PROGRAM P06_LidFeeder
VAR_INPUT
	IbLidFeederDragHomingSensor 			AT %I*  : BOOL;				// Czujnik bazowania
	IbLidFeederDragUpSensor 			 	AT %I*  : BOOL;				// Czujnik
	IbLidFeederDragDownSensor 				AT %I*  : BOOL;				// Czujnik
	IbLidFeederDragLeadBefore1UpSensor 		AT %I*  : BOOL;				// Czujnik
	IbLidFeederUpSensor1 					AT %I*	: BOOL; 								// Czujnik pozycji górnej ssawki podajnika platynek
	IbLidFeederUpSensor2 					AT %I*	: BOOL;
	IbLidFeederDownSensor1 					AT %I*	: BOOL;								
	IbLidFeederDownSensor2 					AT %I*	: BOOL;								
	IbLidFeederLowLevelSensor1  			AT %I* 	: BOOL;	
	IbLidFeederLowLevelSensor2  			AT %I* 	: BOOL;
	IbLidFeederFormPositioning1HideSensor			AT %I*	: BOOL; 
	IbLidFeederFormPositioning2HideSensor			AT %I*	: BOOL;
	IbLidFeederFirstFormSensorBeforeDrag			AT %I*	:BOOL;
	IbLidFeederSuckerSensor 				AT %I*	: BOOL;
	IbLidFeeder2SuckerSensor 				AT %I*	: BOOL;  
	bMovetoEndPositionLidFeeder				:BOOL;	
	QbLidFeederDragActuator                	  		: BOOL;				// Siłownikiem przeciągania (1 faza)					

END_VAR
VAR
	//Podajnik platynek
	fbLidFeeder										: FB_LidFeeder; 						// Blok sterowania podajnikiem platynek
	eLidFeederState									: E_Station; 							// Stan pracy podajnika platynek			
	eLidFeederRunningState							: E_LidFeederState; 					// Stan pracy podajnika platynek
	fbLidFeederState								: FB_State; 

	//Podajnik platynek 2
	fbLidFeeder2									: FB_LidFeeder; 						// Blok sterowania podajnikiem platynek
	eLidFeeder2State								: E_Station; 							// Stan pracy podajnika platynek			
	eLidFeeder2RunningState							: E_LidFeederState; 					// Stan pracy podajnika platynek
	fbLidFeeder2State								: FB_State; 

	QbLidFeederBlockActuator 				AT %Q*	: BOOL;  		// Blokada 
	
	// WEJŚCIA I WYJŚCIA SPRZĘTOWE 1
	QbLidFeeder_FeederActuator1						: BOOL; 				(*Pneu*) 		// Sterowanie zaworem podajnika platynek na wyspie zaworowej
	QbLidFeeder_FeederActuator2						: BOOL; 				(*Pneu*) 		// Sterowanie zaworem podajnika platynek na wyspie zaworowej
	QbLidFeeder_HeaterActuator						: BOOL;  				(*Pneu*) 		// Sterowanie zaworem grzałki platynek na wyspie zaworowej
	QbLidFeeder_SuckerActuator 				AT %Q*	: BOOL; 								// Sterowanie zaworem ssawki platynek na wyspie zaworowej
	QbLidFeederHeaterPWMOut 				AT %Q*	: BOOL; 								// Wyjście sterujące grzałką podajnika platynek
	

	AIbLidFeederHeaterTempCVSensor 			AT %I*	: INT; 									// Wartość aktualnej temperatury grzałki podajnika platynek
	IbLidFeederTempSensorFailure 			AT %I*	: BOOL; 								// Informacja o uszkodzeniu czujnika temperatury grzałki podajnika platynek
	QbLidFeeder_HeightMotorUp 				AT %Q*	: BOOL;									// Sterowanie silnikiem podnosnika stacji w górę 
	QbLidFeeder_HeightMotorDown 			AT %Q*	: BOOL;									//Sterowanie silnikiem podnosnika stacji w dół
	IbLidFeederHeightEncoderPulse  			AT %I* 	: BOOL;									// Wejście impulsów enkodera podnośnika platynek regulacji wysokości 
									// Czujnik niskiego pozimu platynek	
	
	// WEJŚCIA I WYJŚCIA SPRZĘTOWE 2		
	QbLidFeeder2_FeederActuator1					: BOOL; 				(*Pneu*) 		// Sterowanie zaworem podajnika platynek na wyspie zaworowej
	QbLidFeeder2_FeederActuator2					: BOOL; 				(*Pneu*) 		// Sterowanie zaworem podajnika platynek na wyspie zaworowej
	QbLidFeeder2_HeaterActuator						: BOOL;  				(*Pneu*) 		// Sterowanie zaworem grzałki platynek na wyspie zaworowej
	QbLidFeeder2_SuckerActuator 			AT %Q*	: BOOL; 								// Sterowanie zaworem ssawki platynek na wyspie zaworowej
	QbLidFeeder2HeaterPWMOut 				AT %Q*	: BOOL; 								// Wyjście sterujące grzałką podajnika platynek
	IbLidFeeder2UpSensor1 					AT %I*	: BOOL; 								// Czujnik pozycji górnej ssawki podajnika platynek
	IbLidFeeder2DownSensor1 				AT %I*	: BOOL;								
	IbLidFeeder2DownSensor2 				AT %I*	: BOOL;								
									// Czujnik zassania platynki
	AIbLidFeeder2HeaterTempCVSensor 		AT %I*	: INT; 									// Wartość aktualnej temperatury grzałki podajnika platynek
	IbLidFeeder2TempSensorFailure 			AT %I*	: BOOL; 								// Informacja o uszkodzeniu czujnika temperatury grzałki podajnika platynek
										// Czujnik niskiego pozimu platynek
	
	//Vasyl 24.10.25 Aktualizacja enkodera
	IbLidFeederHeightEncoderSetCDone		AT %I*: BOOL;	
	IudiLidFeederHeightEncoderCV         	AT %I*: UDINT; 	
	QbLidFeederHeightEncoderSetC 			AT %Q*: BOOL;		
	QudiLidFeederHeightEncoderSetCV       	AT %Q*: UDINT; 	
	
	tofLidFeederEnable								: TOF;
	tonLidFeederEnable								: TON;
	rtEnable										: R_TRIG;

	tonLidFeederCatchSensorClosed					: TON;
                	
	bTemp											: BOOL;
	bSimulation										: BOOL;
	
	bLidFeederWarning1								: BOOL;
	bLidFeederWarning2								: BOOL;
	
	//PRZECIAGANIE
	eLidFeederDragStation							: E_Station;
	eLidFeederDragRunningStation					: E_DragStationState;
	fbLidFeederDragState							: FB_State;
	fbLidFeederDragStation							: FB_FormsDragStepper;

	tofLidFeederDragStationEnable					: TOF;	
	
	//WEJSCIA I WYJSCIA SPRZETOWE
	QbLidFeederDragLeadBefore1Actuator        		: BOOL;				// Siłownikiem prowadzenia przed 1(1 faza)
	QbLidFeederDragLeadBefore2Actuator        		: BOOL;				// Siłownikiem prowadzenia przed 1(1 faza)
	
	
	IbLidFeederDragLeadBefore2UpSensor 				AT %I*  : BOOL;				// Czujnik
	
	bLidFeederUp									: BOOL;				//Podnoszenie podajników do góry
	
	
	//Chwytak formatek
	fbLidFeederFormPositioning						: FB_Gate;				// Bloczek obsługi bandy
	IbLidFeederFormPositioningUpSensor				AT %I*	: BOOL; 		// 
	QbLidFeederFormPositioningActuator 				: BOOL;  		



	
	bTestManual: BOOL;
END_VAR

//QbLidFeederBlockActuator	:= (GVL.eLidFeederPackageState[1].bFormPresent AND GVL.bFormTransportersDispencerCmdStart) OR 
//							   (GVL.eLidFeederPackageState[2].bFormPresent AND GVL.bFormTransportersDispencerCmdStart);

IF P00_PackML.fbPMLModeManager.eModeStatus = Tc3_PackML.E_PMLUnitMode.ePMLUnitMode_AUTOMATIC AND tofLidFeederEnable.Q THEN
	
	QbLidFeederBlockActuator :=	P00_PackML.fbPMLAuto.ePMLState = Tc3_PackML.E_PMLState.ePMLState_EXECUTE OR 
								P00_PackML.fbPMLAuto.ePMLState = Tc3_PackML.E_PMLState.ePMLState_STOPPING OR 
								P00_PackML.fbPMLAuto.ePMLState = Tc3_PackML.E_PMLState.ePMLState_STARTING;
								
ELSIF P00_PackML.fbPMLModeManager.eModeStatus = Tc3_PackML.E_PMLUnitMode.ePMLUnitMode_MANUAL THEN
	
	QbLidFeederBlockActuator	:= P06_LidSealer.fbLidSealer.bBlockActuator OR P06_LidSealer.fbLidSealer2.bBlockActuator OR VIS.bLidFeeder1ManualHeaterAct OR VIS.bLidFeeder2ManualHeaterAct OR
			VIS.bLidFeeder1Run OR VIS.bLidFeeder2Run OR VIS.bLidFeederEnableShow;
	
END_IF

bLidFeederUp	:= GVL_IO.IbEmergencyStopButton0Pressed OR GVL_IO.IbEmergencyStopButton1Pressed OR GVL_IO.IbEmergencyStopButton2Pressed OR {warning 'PI odkomentować'}
				   GVL_IO.IbEmergencyStopButton3Pressed OR GVL_IO.IbEmergencyStopButton4Pressed OR IbTurnTableEmergencyStopButtonPressed OR (*IbPucksInserterEmergencyStopButton0Pressed OR*) IbPucksInserterEmergencyStopButton1Pressed
				   OR P07_ROPP.IbROPPEmergencyStopButton0Pressed OR P07_ROPP.IbROPPEmergencyStopButton1Pressed 
				AND (QbLidFeeder_HeaterActuator OR QbLidFeeder2_HeaterActuator);
							   
ACT_LidFeeder();
ACT_LidFeeder2();
ACT_LidFeederDragStation();
a_LidFeederFormPositioning();
aLidFeederWarnings();

//GENEROWANIE STANU STACJI DO WIZKI
fbLidFeederState(
	eState 					:= eLidFeederState , 
	bRun 					:= VIS.bLidFeeder1PrepareRun OR VIS.bLidFeeder1Run,	
	eLidFeederRunningState 	:= eLidFeederRunningState , 
	sStateDesc				=> VIS.sLidFeeder1State,
	iState					=> VIS.iLidFeeder1State	);
	
fbLidFeeder2State(
	eState 					:= eLidFeeder2State , 
	bRun 					:= VIS.bLidFeeder2PrepareRun OR VIS.bLidFeeder2Run,	
	eLidFeederRunningState 	:= eLidFeeder2RunningState , 
	sStateDesc				=> VIS.sLidFeeder2State,
	iState					=> VIS.iLidFeeder2State	);
	
(* BAZOWANIE - ZMIAN*)
tonLidFeederEnable(IN := fbLidFeeder.bEnable, PT := T#2S); (*Dodany ton bo Wizka zjebnie wgrywa zmienne, najpierw włacza Enabla a potem dopiero wybiera recepture*)
rtEnable(CLK := tonLidFeederEnable.Q, Q=>);
IF rtEnable.Q AND (P00_PackML.fbPMLAuto.ePMLState = Tc3_PackML.E_PMLState.ePMLState_IDLE OR 
   P00_PackML.fbPMLAuto.ePMLState = Tc3_PackML.E_PMLState.ePMLState_EXECUTE) THEN
    VIS.bLidFeederHeightSet 		:= TRUE;
ELSIF (fbLidFeeder.eState = E_Station.eHomingDone AND fbLidFeeder2.eState = E_Station.eHomingDone)OR VIS.bErrorOccure THEN
    VIS.bLidFeederHeightSet 		:= FALSE;
END_IF
(*KONIEC BAZOWANIE - ZMIANA*)

//PRZEPISYWANIE POMIARÓW
VIS.lrLidFeeder1HeaterTempCV	:= (INT_TO_LREAL(AIbLidFeederHeaterTempCVSensor)/10);
VIS.lrLidFeeder2HeaterTempCV	:= (INT_TO_LREAL(AIbLidFeeder2HeaterTempCVSensor)/10);

//SYMULACJA CZUJNIKÓW IGLIC

//Opoznienie wyłączanie enabla
tofLidFeederEnable(IN:= VIS.bLidFeederEnableShow, PT:=T#2S);

//KASOWANIE ROZKAZÓW CYKLI
IF fbLidFeeder.bCycleDone AND GVL.bManualMode THEN
	VIS.bLidFeeder1PrepareRun 		:= FALSE;
	VIS.bLidFeeder1Run 			:= FALSE;
END_IF
IF fbLidFeeder2.bCycleDone AND GVL.bManualMode THEN
	VIS.bLidFeeder2PrepareRun 		:= FALSE;
	VIS.bLidFeeder2Run 			:= FALSE;
END_IF

IF bSimulation THEN
	IF fbLidFeeder.eState = E_Station.eReady AND fbLidFeeder2.eState = E_Station.eReady THEN
		VIS.bLidFeeder1PrepareRun	:= TRUE;
		VIS.bLidFeeder2PrepareRun	:= TRUE;
	END_IF
	IF fbLidFeeder.eState = E_Station.eRunning AND fbLidFeeder2.eState = E_Station.eRunning THEN
		
		IF (VIS.bLidFeeder1PrepareRun AND NOT VIS.bLidFeeder1Run AND IbLidFeederDownSensor1) AND
		   (VIS.bLidFeeder2PrepareRun AND NOT VIS.bLidFeeder2Run AND IbLidFeeder2DownSensor1) THEN		
			VIS.bLidFeeder1Run 	:= TRUE;
			VIS.bLidFeeder2Run 	:= TRUE;		
	
		END_IF
	END_IF
	
	IF fbLidFeeder.bCycleDone AND fbLidFeeder2.bCycleDone THEN
		
		VIS.bLidFeeder1PrepareRun	:= FALSE;
		VIS.bLidFeeder2PrepareRun	:= FALSE;
		VIS.bLidFeeder1Run 		:= FALSE;
		VIS.bLidFeeder2Run 		:= FALSE;
		
	END_IF
END_IF

(*
{warning: 'Sprawdzic działanie czujnika niskiego poziomu - kiedy stan wysoki'}

//Ostrzeżenia Podajnik 1 
GVL.LidFeederWarning[0].sDescription			:= 'Niski poziom platynek podajnik 1';

IF bLidFeederWarning1 AND NOT GVL.LidFeederWarning[0].bWarning THEN
	
	GVL.LidFeederWarning[0].bWarning			:= TRUE;
	
ELSIF NOT bLidFeederWarning1 AND GVL.LidFeederWarning[0].bAcknowledge THEN
	
	GVL.LidFeederWarning[0].bWarning			:= FALSE;
	GVL.LidFeederWarning[0].bAcknowledge		:= FALSE;
	//GvlVisualization.uliWarningAcknowledge.4 	:= FALSE;
	
ELSIF GVL.LidFeederWarning[0].bAcknowledge THEN
{warning: 'Sprawdzic potwierdzenie warningu tutaj i wewnatrz bloczka gdy zmieni sie stan czujnika '}	
	bLidFeederWarning1							:= FALSE;
	GVL.LidFeederWarning[0].bAcknowledge		:= TRUE;
	
END_IF

//Ostrzeżenia Podajnik 2 
GVL.LidFeederWarning[1].sDescription			:= 'Niski poziom platynek podajnik 2';

IF bLidFeederWarning2 AND NOT GVL.LidFeederWarning[1].bWarning THEN
	
	GVL.LidFeederWarning[1].bWarning			:= TRUE;
	
ELSIF NOT bLidFeederWarning2 AND GVL.LidFeederWarning[1].bAcknowledge THEN
	
	GVL.LidFeederWarning[1].bWarning			:= FALSE;
	GVL.LidFeederWarning[1].bAcknowledge		:= FALSE;
	//GvlVisualization.uliWarningAcknowledge.4 	:= FALSE;
	
ELSIF GVL.LidFeederWarning[1].bAcknowledge THEN
	
	bLidFeederWarning2							:= FALSE;	
	GVL.LidFeederWarning[1].bAcknowledge		:= TRUE;
	
END_IF
*)

//Przeciąganie
tofLidFeederDragStationEnable(IN:= VIS.bLidFeederDragingStationEnableShow, PT:= T#2S);

ACTION a_LidFeederFormPositioning:
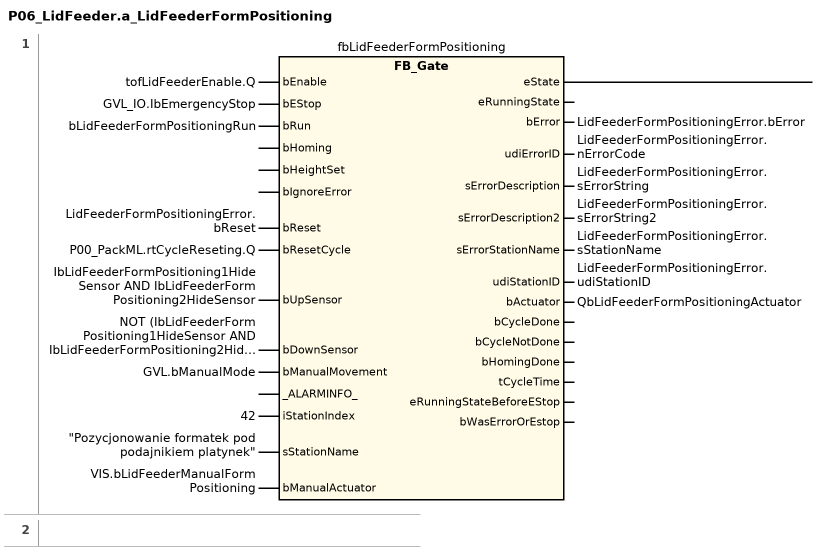
// NETWORK 1
fbLidFeederFormPositioning(
    bEnable := tofLidFeederEnable.Q,
    bEStop := GVL_IO.IbEmergencyStop,
    bRun := bLidFeederFormPositioningRun,
    bReset := LidFeederFormPositioningError.bReset,
    bResetCycle := P00_PackML.rtCycleReseting.Q,
    bUpSensor := IbLidFeederFormPositioning1HideSensor AND IbLidFeederFormPositioning2HideSensor,
    bDownSensor := NOT (IbLidFeederFormPositioning1HideSensor AND IbLidFeederFormPositioning2HideSensor),
    bManualMovement := GVL.bManualMode,
    iStationIndex := 42,
    sStationName := "Pozycjonowanie formatek pod podajnikiem platynek",
    bManualActuator := VIS.bLidFeederManualFormPositioning,
    bError => LidFeederFormPositioningError.bError,
    udiErrorID => LidFeederFormPositioningError.nErrorCode,
    sErrorDescription => LidFeederFormPositioningError.sErrorString,
    sErrorDescription2 => LidFeederFormPositioningError.sErrorString2,
    sErrorStationName => LidFeederFormPositioningError.sStationName,
    udiStationID => LidFeederFormPositioningError.udiStationID,
    bActuator => QbLidFeederFormPositioningActuator); // FB_Gate

// NETWORK 2
END_ACTION

ACTION ACT_LidFeeder:
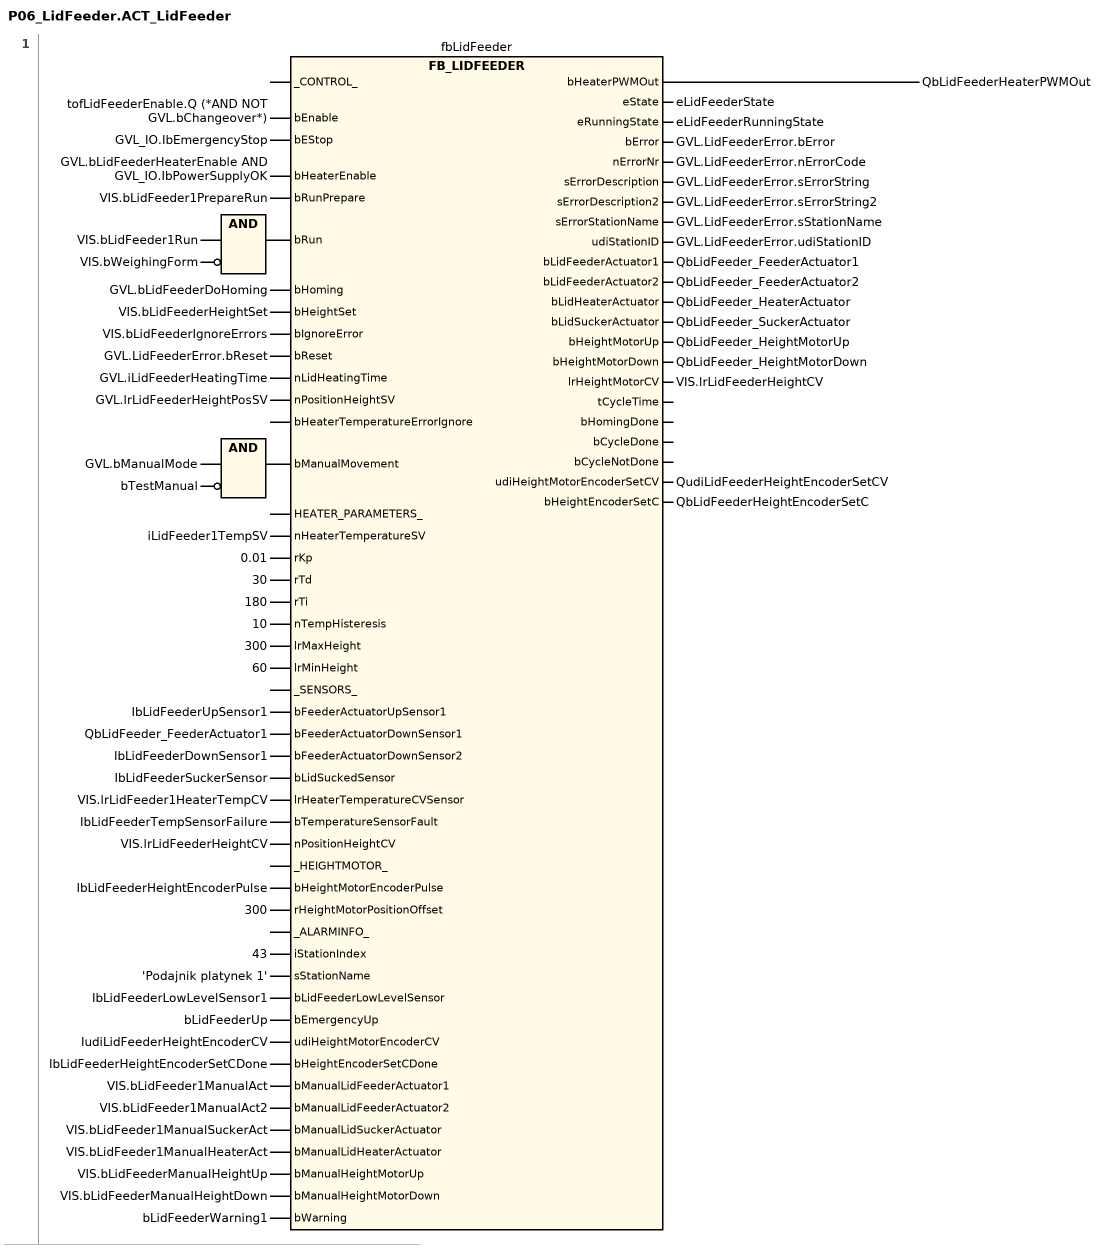
// NETWORK 1
fbLidFeeder(
    bEnable := tofLidFeederEnable.Q (*AND NOT GVL.bChangeover*),
    bEStop := GVL_IO.IbEmergencyStop,
    bHeaterEnable := GVL.bLidFeederHeaterEnable AND GVL_IO.IbPowerSupplyOK,
    bRunPrepare := VIS.bLidFeeder1PrepareRun,
    bRun := VIS.bLidFeeder1Run AND NOT VIS.bWeighingForm,
    bHoming := GVL.bLidFeederDoHoming,
    bHeightSet := VIS.bLidFeederHeightSet,
    bIgnoreError := VIS.bLidFeederIgnoreErrors,
    bReset := GVL.LidFeederError.bReset,
    nLidHeatingTime := GVL.iLidFeederHeatingTime,
    nPositionHeightSV := GVL.lrLidFeederHeightPosSV,
    bManualMovement := GVL.bManualMode AND NOT bTestManual,
    nHeaterTemperatureSV := iLidFeeder1TempSV,
    rKp := 0.01,
    rTd := 30,
    rTi := 180,
    nTempHisteresis := 10,
    lrMaxHeight := 300,
    lrMinHeight := 60,
    bFeederActuatorUpSensor1 := IbLidFeederUpSensor1,
    bFeederActuatorDownSensor1 := QbLidFeeder_FeederActuator1,
    bFeederActuatorDownSensor2 := IbLidFeederDownSensor1,
    bLidSuckedSensor := IbLidFeederSuckerSensor,
    lrHeaterTemperatureCVSensor := VIS.lrLidFeeder1HeaterTempCV,
    bTemperatureSensorFault := IbLidFeederTempSensorFailure,
    nPositionHeightCV := VIS.lrLidFeederHeightCV,
    bHeightMotorEncoderPulse := IbLidFeederHeightEncoderPulse,
    rHeightMotorPositionOffset := 300,
    iStationIndex := 43,
    sStationName := 'Podajnik platynek 1',
    bLidFeederLowLevelSensor := IbLidFeederLowLevelSensor1,
    bEmergencyUp := bLidFeederUp,
    udiHeightMotorEncoderCV := IudiLidFeederHeightEncoderCV,
    bHeightEncoderSetCDone := IbLidFeederHeightEncoderSetCDone,
    bManualLidFeederActuator1 := VIS.bLidFeeder1ManualAct,
    bManualLidFeederActuator2 := VIS.bLidFeeder1ManualAct2,
    bManualLidSuckerActuator := VIS.bLidFeeder1ManualSuckerAct,
    bManualLidHeaterActuator := VIS.bLidFeeder1ManualHeaterAct,
    bManualHeightMotorUp := VIS.bLidFeederManualHeightUp,
    bManualHeightMotorDown := VIS.bLidFeederManualHeightDown,
    bWarning := bLidFeederWarning1,
    eState => eLidFeederState,
    eRunningState => eLidFeederRunningState,
    bError => GVL.LidFeederError.bError,
    nErrorNr => GVL.LidFeederError.nErrorCode,
    sErrorDescription => GVL.LidFeederError.sErrorString,
    sErrorDescription2 => GVL.LidFeederError.sErrorString2,
    sErrorStationName => GVL.LidFeederError.sStationName,
    udiStationID => GVL.LidFeederError.udiStationID,
    bLidFeederActuator1 => QbLidFeeder_FeederActuator1,
    bLidFeederActuator2 => QbLidFeeder_FeederActuator2,
    bLidHeaterActuator => QbLidFeeder_HeaterActuator,
    bLidSuckerActuator => QbLidFeeder_SuckerActuator,
    bHeightMotorUp => QbLidFeeder_HeightMotorUp,
    bHeightMotorDown => QbLidFeeder_HeightMotorDown,
    lrHeightMotorCV => VIS.lrLidFeederHeightCV,
    udiHeightMotorEncoderSetCV => QudiLidFeederHeightEncoderSetCV,
    bHeightEncoderSetC => QbLidFeederHeightEncoderSetC); // FB_LIDFEEDER
QbLidFeederHeaterPWMOut := fbLidFeeder.bHeaterPWMOut;
END_ACTION

ACTION ACT_LidFeeder2:
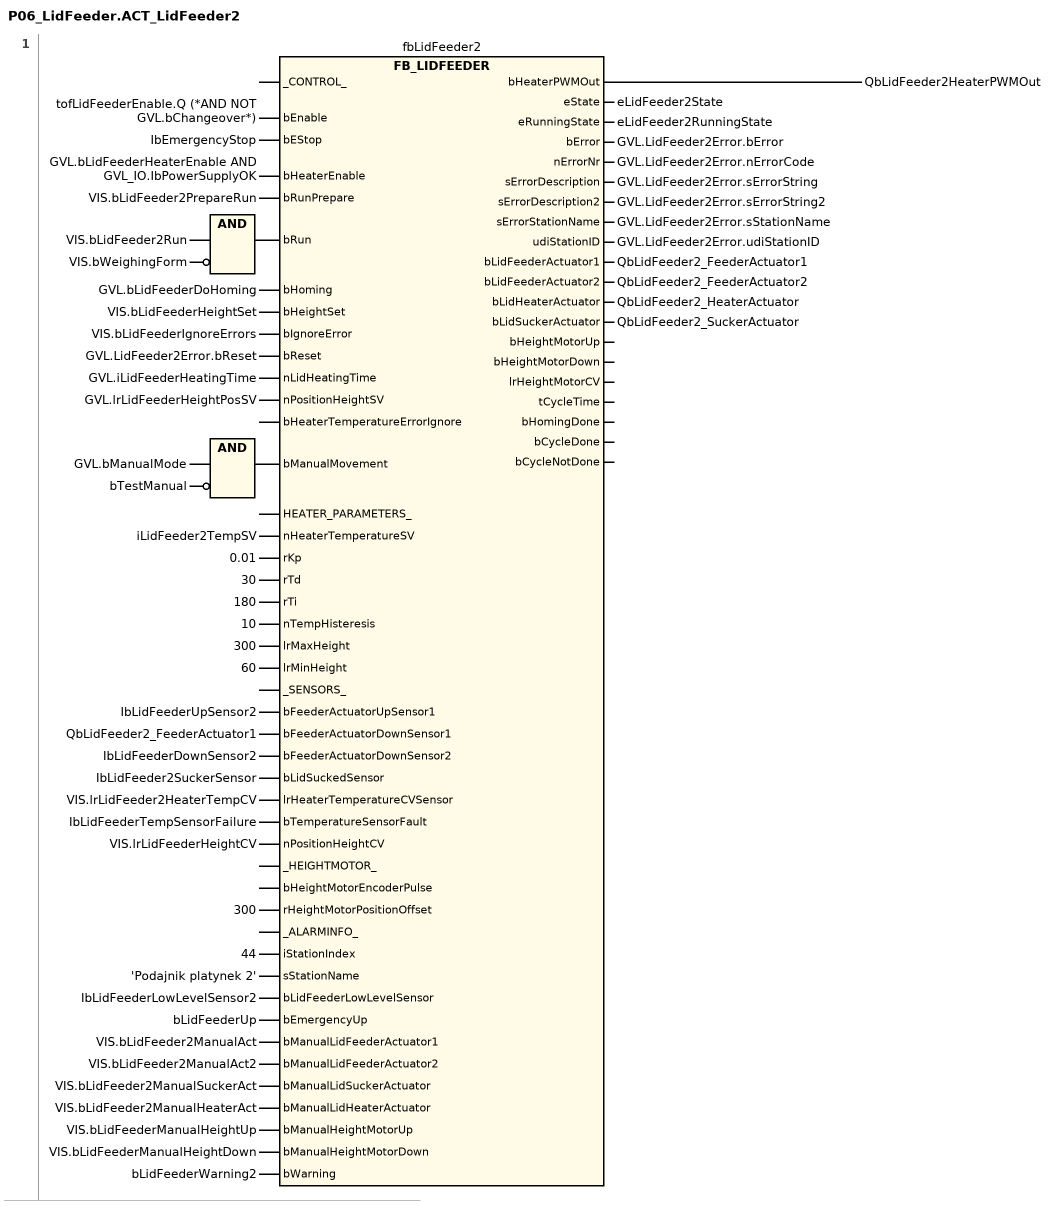
// NETWORK 1
fbLidFeeder2(
    bEnable := tofLidFeederEnable.Q (*AND NOT GVL.bChangeover*),
    bEStop := IbEmergencyStop,
    bHeaterEnable := GVL.bLidFeederHeaterEnable AND GVL_IO.IbPowerSupplyOK,
    bRunPrepare := VIS.bLidFeeder2PrepareRun,
    bRun := VIS.bLidFeeder2Run AND NOT VIS.bWeighingForm,
    bHoming := GVL.bLidFeederDoHoming,
    bHeightSet := VIS.bLidFeederHeightSet,
    bIgnoreError := VIS.bLidFeederIgnoreErrors,
    bReset := GVL.LidFeeder2Error.bReset,
    nLidHeatingTime := GVL.iLidFeederHeatingTime,
    nPositionHeightSV := GVL.lrLidFeederHeightPosSV,
    bManualMovement := GVL.bManualMode AND NOT bTestManual,
    nHeaterTemperatureSV := iLidFeeder2TempSV,
    rKp := 0.01,
    rTd := 30,
    rTi := 180,
    nTempHisteresis := 10,
    lrMaxHeight := 300,
    lrMinHeight := 60,
    bFeederActuatorUpSensor1 := IbLidFeederUpSensor2,
    bFeederActuatorDownSensor1 := QbLidFeeder2_FeederActuator1,
    bFeederActuatorDownSensor2 := IbLidFeederDownSensor2,
    bLidSuckedSensor := IbLidFeeder2SuckerSensor,
    lrHeaterTemperatureCVSensor := VIS.lrLidFeeder2HeaterTempCV,
    bTemperatureSensorFault := IbLidFeederTempSensorFailure,
    nPositionHeightCV := VIS.lrLidFeederHeightCV,
    rHeightMotorPositionOffset := 300,
    iStationIndex := 44,
    sStationName := 'Podajnik platynek 2',
    bLidFeederLowLevelSensor := IbLidFeederLowLevelSensor2,
    bEmergencyUp := bLidFeederUp,
    bManualLidFeederActuator1 := VIS.bLidFeeder2ManualAct,
    bManualLidFeederActuator2 := VIS.bLidFeeder2ManualAct2,
    bManualLidSuckerActuator := VIS.bLidFeeder2ManualSuckerAct,
    bManualLidHeaterActuator := VIS.bLidFeeder2ManualHeaterAct,
    bManualHeightMotorUp := VIS.bLidFeederManualHeightUp,
    bManualHeightMotorDown := VIS.bLidFeederManualHeightDown,
    bWarning := bLidFeederWarning2,
    eState => eLidFeeder2State,
    eRunningState => eLidFeeder2RunningState,
    bError => GVL.LidFeeder2Error.bError,
    nErrorNr => GVL.LidFeeder2Error.nErrorCode,
    sErrorDescription => GVL.LidFeeder2Error.sErrorString,
    sErrorDescription2 => GVL.LidFeeder2Error.sErrorString2,
    sErrorStationName => GVL.LidFeeder2Error.sStationName,
    udiStationID => GVL.LidFeeder2Error.udiStationID,
    bLidFeederActuator1 => QbLidFeeder2_FeederActuator1,
    bLidFeederActuator2 => QbLidFeeder2_FeederActuator2,
    bLidHeaterActuator => QbLidFeeder2_HeaterActuator,
    bLidSuckerActuator => QbLidFeeder2_SuckerActuator); // FB_LIDFEEDER
QbLidFeeder2HeaterPWMOut := fbLidFeeder2.bHeaterPWMOut;
END_ACTION

ACTION ACT_LidFeederDragStation:
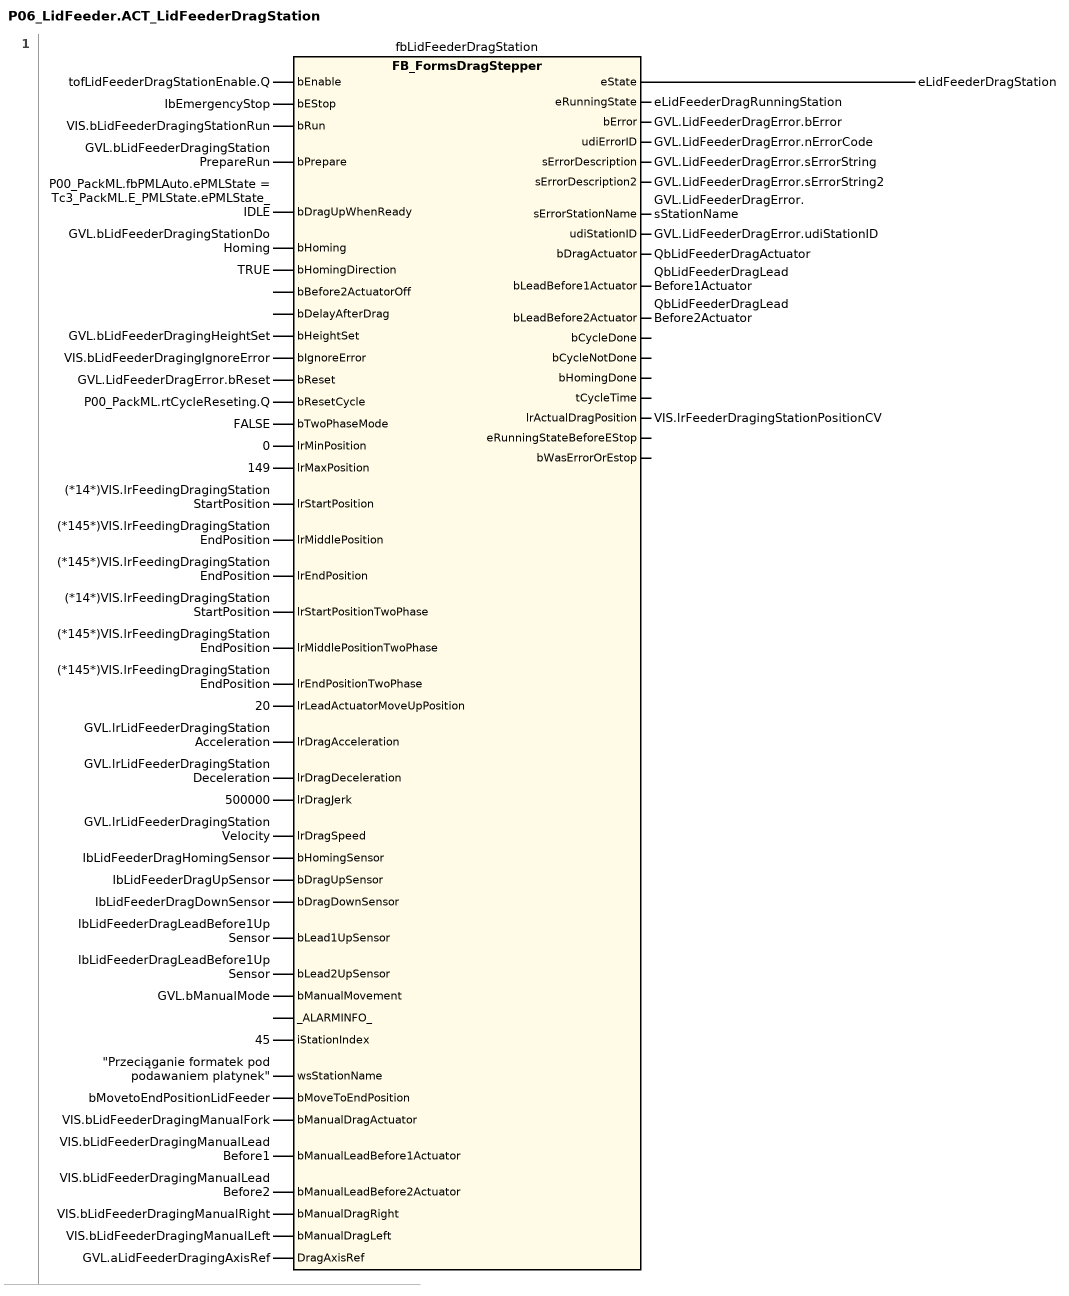
// NETWORK 1
fbLidFeederDragStation(
    bEnable := tofLidFeederDragStationEnable.Q,
    bEStop := IbEmergencyStop,
    bRun := VIS.bLidFeederDragingStationRun,
    bPrepare := GVL.bLidFeederDragingStationPrepareRun,
    bDragUpWhenReady := P00_PackML.fbPMLAuto.ePMLState = Tc3_PackML.E_PMLState.ePMLState_IDLE,
    bHoming := GVL.bLidFeederDragingStationDoHoming,
    bHomingDirection := TRUE,
    bHeightSet := GVL.bLidFeederDragingHeightSet,
    bIgnoreError := VIS.bLidFeederDragingIgnoreError,
    bReset := GVL.LidFeederDragError.bReset,
    bResetCycle := P00_PackML.rtCycleReseting.Q,
    bTwoPhaseMode := FALSE,
    lrMinPosition := 0,
    lrMaxPosition := 149,
    lrStartPosition := (*14*)VIS.lrFeedingDragingStationStartPosition,
    lrMiddlePosition := (*145*)VIS.lrFeedingDragingStationEndPosition,
    lrEndPosition := (*145*)VIS.lrFeedingDragingStationEndPosition,
    lrStartPositionTwoPhase := (*14*)VIS.lrFeedingDragingStationStartPosition,
    lrMiddlePositionTwoPhase := (*145*)VIS.lrFeedingDragingStationEndPosition,
    lrEndPositionTwoPhase := (*145*)VIS.lrFeedingDragingStationEndPosition,
    lrLeadActuatorMoveUpPosition := 20,
    lrDragAcceleration := GVL.lrLidFeederDragingStationAcceleration,
    lrDragDeceleration := GVL.lrLidFeederDragingStationDeceleration,
    lrDragJerk := 500000,
    lrDragSpeed := GVL.lrLidFeederDragingStationVelocity,
    bHomingSensor := IbLidFeederDragHomingSensor,
    bDragUpSensor := IbLidFeederDragUpSensor,
    bDragDownSensor := IbLidFeederDragDownSensor,
    bLead1UpSensor := IbLidFeederDragLeadBefore1UpSensor,
    bLead2UpSensor := IbLidFeederDragLeadBefore1UpSensor,
    bManualMovement := GVL.bManualMode,
    iStationIndex := 45,
    wsStationName := "Przeciąganie formatek pod podawaniem platynek",
    bMoveToEndPosition := bMovetoEndPositionLidFeeder,
    bManualDragActuator := VIS.bLidFeederDragingManualFork,
    bManualLeadBefore1Actuator := VIS.bLidFeederDragingManualLeadBefore1,
    bManualLeadBefore2Actuator := VIS.bLidFeederDragingManualLeadBefore2,
    bManualDragRight := VIS.bLidFeederDragingManualRight,
    bManualDragLeft := VIS.bLidFeederDragingManualLeft,
    DragAxisRef := GVL.aLidFeederDragingAxisRef,
    eRunningState => eLidFeederDragRunningStation,
    bError => GVL.LidFeederDragError.bError,
    udiErrorID => GVL.LidFeederDragError.nErrorCode,
    sErrorDescription => GVL.LidFeederDragError.sErrorString,
    sErrorDescription2 => GVL.LidFeederDragError.sErrorString2,
    sErrorStationName => GVL.LidFeederDragError.sStationName,
    udiStationID => GVL.LidFeederDragError.udiStationID,
    bDragActuator => QbLidFeederDragActuator,
    bLeadBefore1Actuator => QbLidFeederDragLeadBefore1Actuator,
    bLeadBefore2Actuator => QbLidFeederDragLeadBefore2Actuator,
    lrActualDragPosition => VIS.lrFeederDragingStationPositionCV); // FB_FormsDragStepper
eLidFeederDragStation := fbLidFeederDragStation.eState;
END_ACTION

ACTION ACT_Limits:
(*
Nazwa:			aSetRecipe
Opis:			Zapisywanie zmiennych gdy mają wartość 0 
Wersja:			v0.1
Data:			2022-06-22
Autor:			DP
Urzadzenia:		
Konfiguracja:	
Info:
- zabezpieczenie przed recepturami które nie mają tych parametrów i jest w nich wartość 0
*)

IF 	VIS.lrFeedingDragingStationStartPosition		= 0		THEN	VIS.lrFeedingDragingStationStartPosition		:=	14;		END_IF;
IF 	VIS.lrFeedingDragingStationEndPosition		= 0		THEN	VIS.lrFeedingDragingStationEndPosition		:=	145;	END_IF;
END_ACTION

ACTION aLidFeederWarnings:

//Warning 0
LidFeederWarning[0].sDescription:='Podajnik platynek 1 | Brak platynek w zasobniku';
IF bLidFeederWarning1 AND NOT LidFeederWarning[0].bWarning AND bLidFeederEnable THEN
	LidFeederWarning[0].bWarning:=TRUE;
ELSIF NOT bLidFeederWarning1 AND LidFeederWarning[0].bAcknowledge THEN
	LidFeederWarning[0].bWarning		:=	FALSE;
	LidFeederWarning[0].bAcknowledge	:=	FALSE;
	VIS.uliWarningOccure.39				:=	FALSE;
ELSIF LidFeederWarning[0].bAcknowledge THEN
	LidFeederWarning[0].bAcknowledge	:=	TRUE;
END_IF

//Warning 1
LidFeederWarning[1].sDescription:='Podajnik platynek 2 | Brak platynek w zasobniku';
IF bLidFeederWarning2 AND NOT LidFeederWarning[1].bWarning AND bLidFeederEnable THEN
	LidFeederWarning[1].bWarning:=TRUE;
ELSIF NOT bLidFeederWarning2 AND LidFeederWarning[1].bAcknowledge THEN
	LidFeederWarning[1].bWarning		:=	FALSE;
	LidFeederWarning[1].bAcknowledge	:=	FALSE;
	VIS.uliWarningOccure.40				:=	FALSE;
ELSIF LidFeederWarning[1].bAcknowledge THEN
	LidFeederWarning[1].bAcknowledge	:=	TRUE;
END_IF
END_ACTION

END_PROGRAM

(* stored: Version 1.1.0.1, ProductVersion 3.1.4026.13, FileIdentifier 7e56a2bf735942a56fadfc51384c7ca9cf95543b, FileSignature 86a622c485db353d401428cbe6fa96b066f8de3d2cdf8b75f2381994092af08a664668a7bdfaafdeb639efe79a4961be2e708a795b63138e3e61dc6b6ad6ed15a127413051a21345f68742a4bf06715331e1608eb0d2c26237d27d08af7eadf16f8bd5a38b7573ccc207bcc854ac169034d39adab9beebc4108f72eeb1e6c91a22f71c5b160952e190c7ff25ee414ed9ddb85faec58686fcf92d469588eae4777423564036f7172233650f3ea1518d7083cb7e9f4d44ee35fccdb01fdcea1770a31781bb0b0d63ea02a6f87bda8ae3d9e40156c9cc7a4139dee94772a32d521d40aba182db3af21bbd34cfea3a7507bbf13aca1f1bba49349022185d70096e85
   POU P06_LidFeeder: Id {5f4fd25a-7185-4e71-be43-ffd96a7f327d}, SpecialFunc None
   Action a_LidFeederFormPositioning: Id {b74e8c26-cded-4f93-9403-b9899b33fa91}
   Action ACT_LidFeeder: Id {c93f8fff-510a-4216-9b42-f88d49bb5148}
   Action ACT_LidFeeder2: Id {afe372ef-057d-4108-80c8-fe32f6e566cc}
   Action ACT_LidFeederDragStation: Id {9900aaa8-e6a8-462b-92f9-d5552208140b}
   Action ACT_Limits: Id {1c6cfa10-b677-4e2d-b137-9bbb0f15ec0e}
   Action aLidFeederWarnings: Id {285c0428-303d-4831-b06f-906476cf8dee} *)
